(* LS Electric XG5000 project: AABB *)
(* PLC LSPLC *)

PROGRAM NewProgram (* task: Scan Program *)
VAR
    Control AT %QX0.0.0 : BOOL;
    Control_1 AT %QX0.0.1 : BOOL;
    Counter_1 : BOOL;
    Flag : BOOL;
    Flag_1 : BOOL;
    Load_Posative_A : BOOL;
    PBS_1 AT %IX0.0.1 : BOOL;
    PBS_2 AT %IX0.0.3 : BOOL;
    PBS_3 AT %IX0.0.2 : BOOL;
    PBS_4 AT %IX0.0.4 : BOOL;
END_VAR

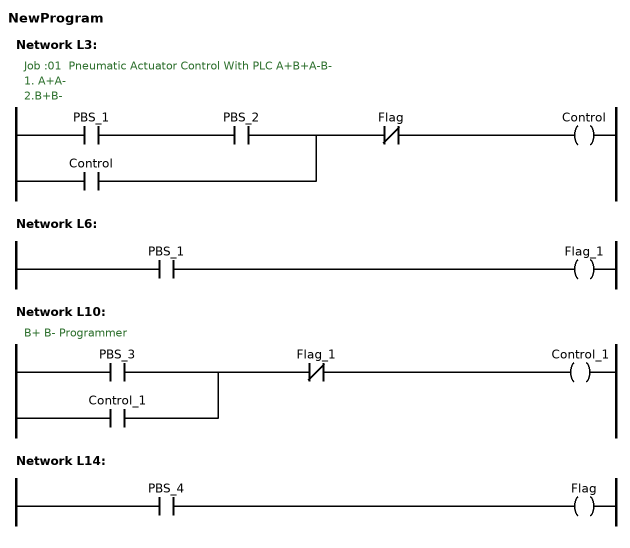
(* Job :01  Pneumatic Actuator Control With PLC A+B+A-B- *)
(* 1. A+A- *)
(* 2.B+B- *)
(* Rung L3 *)
Control := ((PBS_1 AND PBS_2) OR Control) AND NOT Flag;
(* Rung L6 *)
Flag_1 := PBS_1;
(* B+ B- Programmer *)
(* Rung L10 *)
Control_1 := (PBS_3 OR Control_1) AND NOT Flag_1;
(* Rung L14 *)
Flag := PBS_4;
END_PROGRAM